// TIA Portal V16 export
// export: Created 2024-09-05T17:40:14.2364579Z, ExportSetting WithDefaults, DisplayName Totally Integrated Automation Portal, DisplayVersion V16 Update 6, DisplayName TIA Portal Version Control Interface, DisplayVersion V16 Update 2, DisplayName TIA Portal Openness, DisplayVersion V16 Update 6, DisplayName STEP 7 Professional, DisplayVersion V16 Update 6, DisplayName STEP 7 Safety, DisplayVersion V16, DisplayName WinCC Advanced, DisplayVersion V16 Update 6
TYPE "UDT_TurnTable"
// stored: IsFailsafeCompliant false
   STRUCT
      Commands : Struct
         ManualMode : "UDT_TurnTableCommands";
         AutomaticMode { S7_SetPoint := 'True'} : "UDT_TurnTableCommands";
      END_STRUCT;
      Status : "UDT_TurnTableStatus";
      "I/O" { S7_SetPoint := 'True'} : "UDT_TurnTable_I/O";
   END_STRUCT;
END_TYPE
